DATA_BLOCK "ID_Plate_CM_DI_iPlateSenCilPushingIn_d0"
{ S7_Optimized_Access := 'FALSE' }
VERSION : 0.1
NON_RETAIN
"FB_CM_DI_Sensor"

BEGIN

END_DATA_BLOCK

